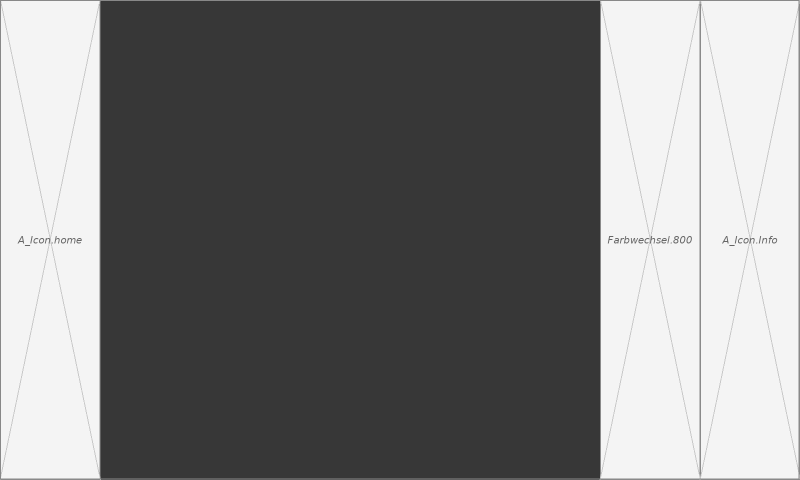
VISUALIZATION Sollwertmenu  // 800x480
    Frame (0,0 800x430)
        shows GWP_Library.Sollwertmenu()
    Frame (0,55 800x121)
        shows GWP_Library.Kachel_Solwertmenu_WG()
        OnMouseClick: change screen: Sollwertmenu_Waermegewinnung
    Frame (0,180 800x121)
        shows GWP_Library.Kachel_Solwertmenu_WP()
        OnMouseClick: change screen: Sollwertmenu_Waermepumpe
    Frame (0,305 800x121)
        shows GWP_Library.Kachel_Solwertmenu_WS()
        OnMouseClick: change screen: Sollwertmenu_Waermesenke
    Frame (0,0 800x480)
        shows Fusszeile_50()
END_VISUALIZATION

// ---- VISUs/Sollwertmenu/Sollwertmenu_Zirk_PU.TcVIS
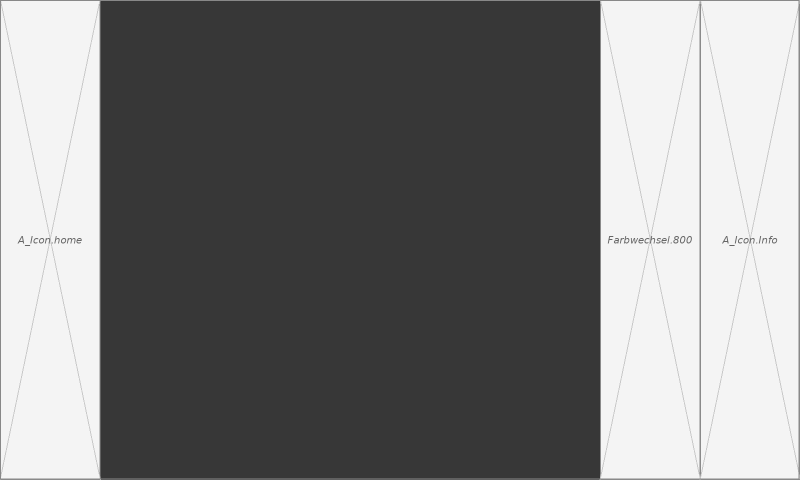
VISUALIZATION Sollwertmenu_Zirk_PU  // 800x480
    Frame (0,0 800x430)
        shows GWP_Library.Sollwertmenu_Zirk_PU()
    Frame (0,55 398x122)
        shows GWP_Library.Kachel_Zirk_PU()
        OnMouseClick: change screen: Zirkulationspumpe_Sollwerte
    Frame (402,55 398x122)
        shows GWP_Library.Kachel_Zirk_PU_Wochenuhr()
        OnMouseClick: change screen: Zirkulationspumpe_CLK_W7_Siebentageprogramm
    Frame (0,0 800x480)
        shows Fusszeile_50()
END_VISUALIZATION

// ---- VISUs/Sollwertmenu/Sollwertmenu_Waermegewinnung.TcVIS
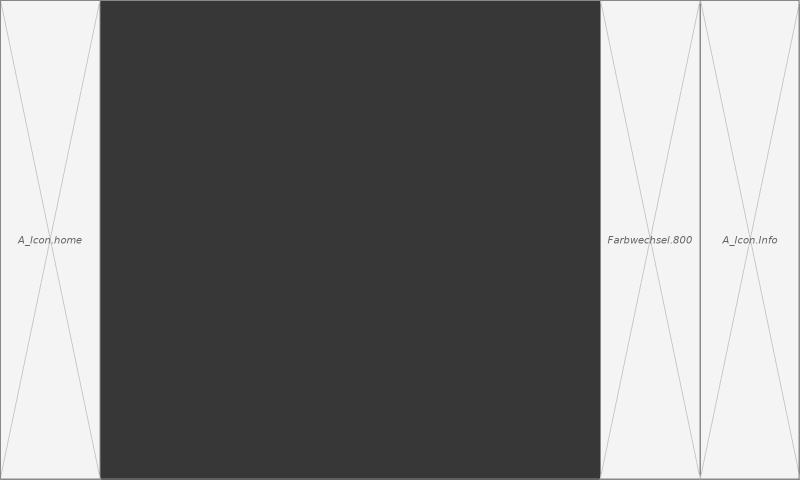
VISUALIZATION Sollwertmenu_Waermegewinnung  // 800x480
    Frame (0,0 800x430)
        shows GWP_Library.Sollwertmenu_Waermegewinnung(FB_KWP_SP_AC_NC := Main.KWP_SP_AC_NC_0, FB_Kreis_3KO := Main.Kreis_3KO_0)
    Frame (0,55 398x121)
        shows GWP_Library.Kachel_PU_VD()
        OnMouseClick: change screen: VD_PU_Sollwerte
    Frame (402,55 398x121)
        shows GWP_Library.Kachel_PU_GW()
        OnMouseClick: change screen: VD_GW_Sollwerte
    Frame (0,304 398x121)
        shows GWP_Library.Kachel_Kaltwasser(FB_Kreis_3KO := Main.Kreis_3KO_0)
        OnMouseClick: change screen: Sollwertmenu_KWP
    Frame (402,179 398x121)
        shows GWP_Library.Kachel_KD_Sollwerte_zuruecksetzen()
        OnMouseClick: change screen: VD_Sollwerte_zuruecksetzen
    Frame (0,179 398x121)
        shows GWP_Library.Kachel_VD_VTL()
        OnMouseClick: change screen: VD_VTL_Sollwerte
    Frame (0,0 800x480)
        shows Fusszeile_50()
END_VISUALIZATION

// ---- VISUs/Sollwertmenu/Sollwertmenu_Waermepumpe.TcVIS
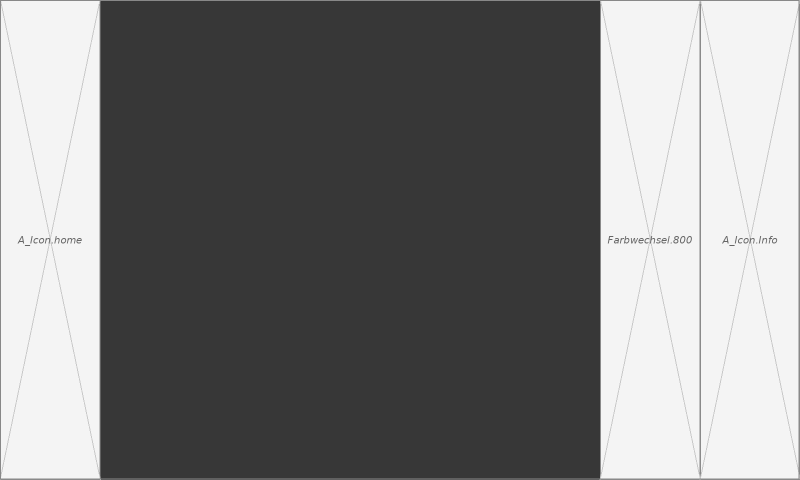
VISUALIZATION Sollwertmenu_Waermepumpe  // 800x480
    Frame (0,0 800x430)
        shows GWP_Library.Sollwertmenu_Waermepumpe()
    Frame (402,55 398x121)
        shows GWP_Library.Kachel_EEV()
        OnMouseClick: change screen: EEv
    Frame (0,179 398x121)
        shows GWP_Library.Kachel_Einsatzgrenzen()
        OnMouseClick: change screen: EG_Innen
    Frame (0,55 398x121)
        shows GWP_Library.Kachel_Allgemein_WP()
        OnMouseClick: change screen: Kreis_3KO_SollwerteAllg
    Frame (0,0 800x480)
        shows Fusszeile_50()
END_VISUALIZATION

// ---- VISUs/Sollwertmenu/Sollwertmenu_KWP.TcVIS
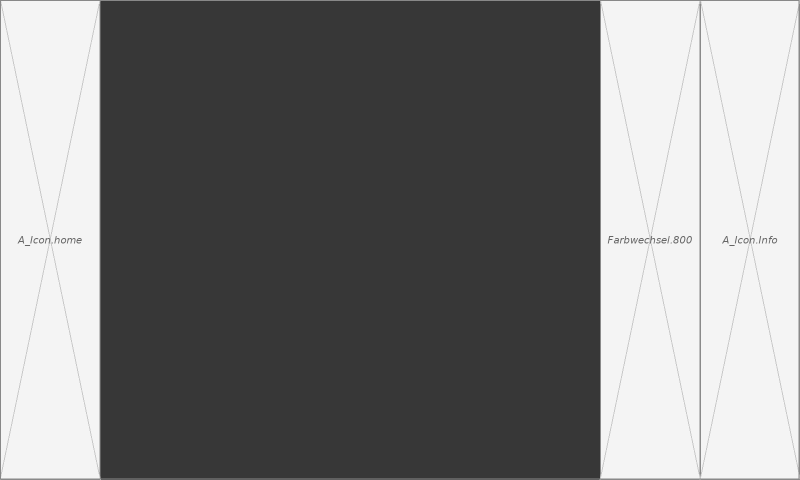
VISUALIZATION Sollwertmenu_KWP  // 800x480
    Frame (0,0 800x430)
        shows GWP_Library.Sollwertmenu_KWP()
    Frame (0,55 398x122)
        shows GWP_Library.Kachel_KWP_Sollwerte(FB_Kreis_3KO := Main.Kreis_3KO_0)
        OnMouseClick: change screen: KWP_SP_AC_NC_Sollwerte
    Frame (402,55 398x122)
        shows GWP_Library.Kachel_KWP_Pumpe()
        OnMouseClick: change screen: KWP_SP_AC_NC_PU_Sollwerte
    Frame (0,179 398x122)
        shows GWP_Library.Kachel_KWP_Tagesuhr_Kuehlkurve()
        OnMouseClick: change screen: KWP_SP_AC_NC_CLK_D
    Frame (402,179 398x121)
        shows GWP_Library.Kachel_KWP_Kuehlkurve()
        OnMouseClick: change screen: KWP_SP_AC_NC_GR_4_ohne_RE
    Frame (0,0 800x480)
        shows Fusszeile_50()
END_VISUALIZATION

// ---- VISUs/Sollwertmenu/Sollwertmenu_Waermesenke.TcVIS
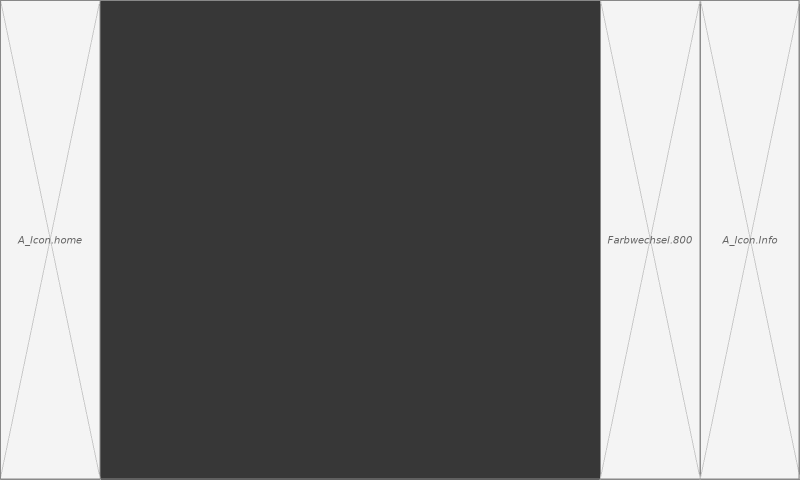
VISUALIZATION Sollwertmenu_Waermesenke  // 800x480
    Frame (0,0 800x430)
        shows GWP_Library.Sollwertmenu_Waermesenke()
    Frame (0,55 398x121)
        shows GWP_Library.Kachel_Hochhaltung()
        OnMouseClick: change screen: Sollwertmenu_KD
    Frame (402,55 398x121)
        shows GWP_Library.Kachel_HWP()
        OnMouseClick: change screen: Sollwertmenu_HWP
    Frame (0,179 398x121)
        shows GWP_Library.Kachel_TWW()
        OnMouseClick: change screen: Sollwertmenu_TWW
    Frame (402,179 398x121)
        shows GWP_Library.Kachel_Zusatzheitzung()
        OnMouseClick: change screen: Zusatzheizung_Sollwerte
    Frame (0,303 398x121)
        shows GWP_Library.Kachel_Zirk_Pumpe()
        OnMouseClick: change screen: Sollwertmenu_Zirk_PU
    Frame (0,55 398x121)
        shows GWP_Library.Kachel_Hochhaltung()
        OnMouseClick: change screen: Sollwertmenu_KD
    Frame (402,55 398x121)
        shows GWP_Library.Kachel_HWP()
        OnMouseClick: change screen: Sollwertmenu_HWP
    Frame (0,179 398x121)
        shows GWP_Library.Kachel_TWW()
        OnMouseClick: change screen: Sollwertmenu_TWW
    Frame (402,179 398x121)
        shows GWP_Library.Kachel_Zirk_PU()
        OnMouseClick: change screen: Sollwertmenu_Zirk_PU
    Frame (0,303 398x121)
        shows GWP_Library.Kachel_Zusatzheitzung()
        OnMouseClick: change screen: Zusatzheizung_Sollwerte
    Frame (0,0 800x480)
        shows Fusszeile_50()
END_VISUALIZATION

// ---- VISUs/Sollwertmenu/Sollwertmenu_KD.TcVIS
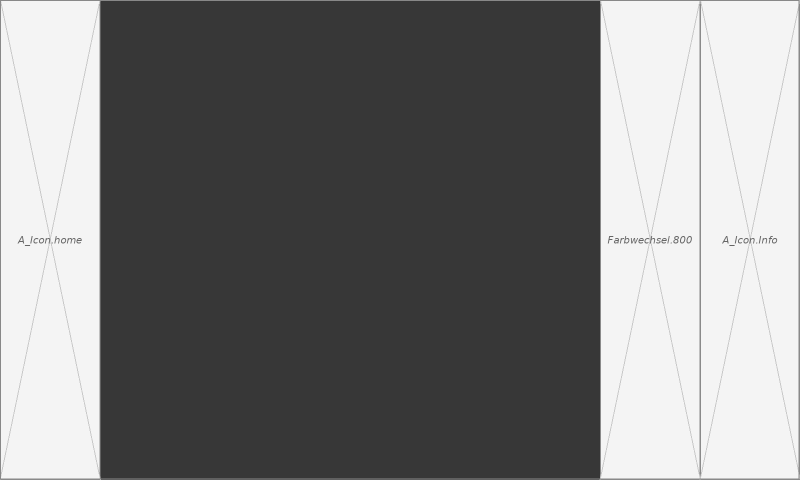
VISUALIZATION Sollwertmenu_KD  // 800x480
    Frame (0,0 800x430)
        shows GWP_Library.Sollwertmenu_KD()
    Frame (0,55 398x121)
        shows GWP_Library.Kachel_KD_Pumpe()
        OnMouseClick: change screen: KD_PU_Sollwerte
    Frame (402,55 398x121)
        shows GWP_Library.Kachel_KD_Ventil()
        OnMouseClick: change screen: KD_VTL_Sollwerte
    Frame (0,179 398x121)
        shows GWP_Library.Kachel_KD_Sollwerte_zuruecksetzen()
        OnMouseClick: change screen: KD_Sollwerte_zuruecksetzen
    Frame (0,0 800x480)
        shows Fusszeile_50()
END_VISUALIZATION

// ---- VISUs/Sollwertmenu/Sollwertmenu_HWP.TcVIS
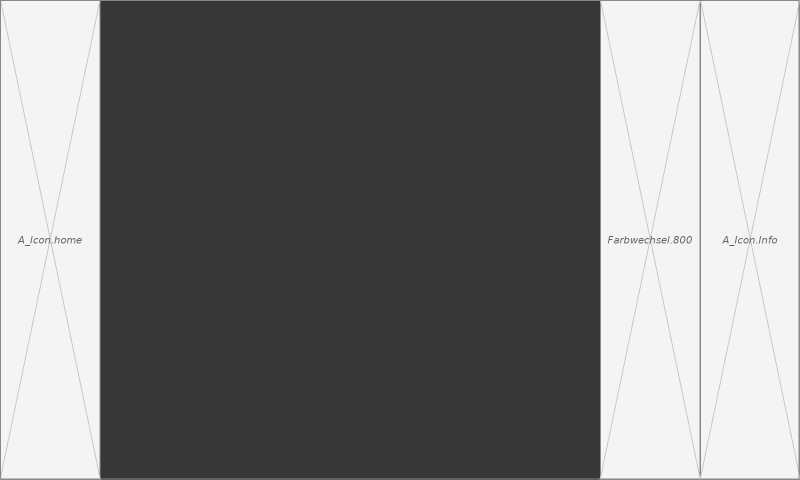
VISUALIZATION Sollwertmenu_HWP  // 800x480
    Frame (0,0 800x430)
        shows GWP_Library.Sollwertmenu_HWP()
    Frame (0,55 398x121)
        shows GWP_Library.Kachel_HWP_Sollwerte(FB_Kreis_3KO := Main.Kreis_3KO_0)
        OnMouseClick: change screen: HWP_SP_Sollwerte
    Frame (402,55 398x121)
        shows GWP_Library.Kachel_HWP_Tagesuhr_Heizkurve()
        OnMouseClick: change screen: HWP_SP_CLK_D
    Frame (0,179 398x121)
        shows GWP_Library.Kachel_HWP_Heizkurve()
        OnMouseClick: change screen: HWP_SP_GR_4_ohne_RE
    Frame (0,0 800x480)
        shows Fusszeile_50()
END_VISUALIZATION

// ---- VISUs/Sollwertmenu/Sollwertmenu_TWW.TcVIS
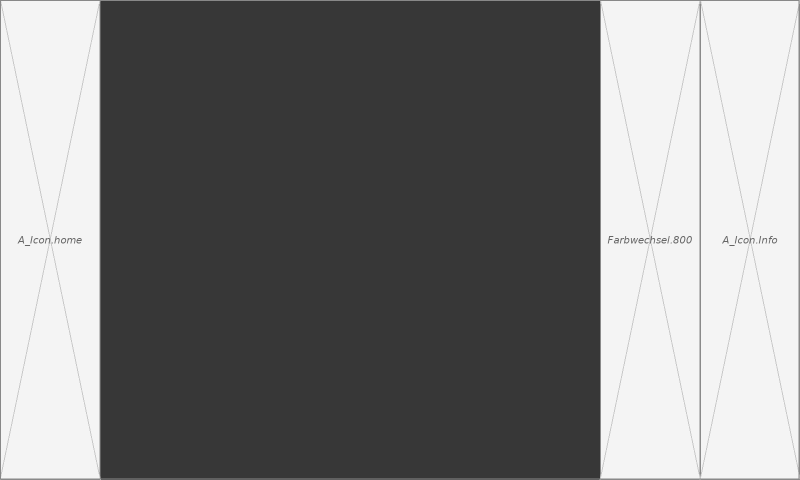
VISUALIZATION Sollwertmenu_TWW  // 800x480
    Frame (0,0 800x430)
        shows GWP_Library.Sollwertmenu_TWW()
    Frame (0,55 398x121)
        shows GWP_Library.Kachel_TWW_SP_Sollwerte()
        OnMouseClick: change screen: TWW_SP_Sollwerte
    Frame (402,55 398x121)
        shows GWP_Library.Kachel_TWW_SP_Pumpe()
        OnMouseClick: change screen: TWW_SP_PU_Sollwerte
    Frame (0,179 398x121)
        shows GWP_Library.Kachel_TWW_SP_Zwangsladung_1()
        OnMouseClick: change screen: TWW_SP_CLK_I_Zwangsladung_1
    Frame (402,179 398x121)
        shows GWP_Library.Kachel_TWW_SP_Zwangsladung_2()
        OnMouseClick: change screen: TWW_SP_CLK_I_Zwangsladung_2
    Frame (0,0 800x480)
        shows Fusszeile_50()
END_VISUALIZATION

// ---- VISUs/Test_Login.TcVIS
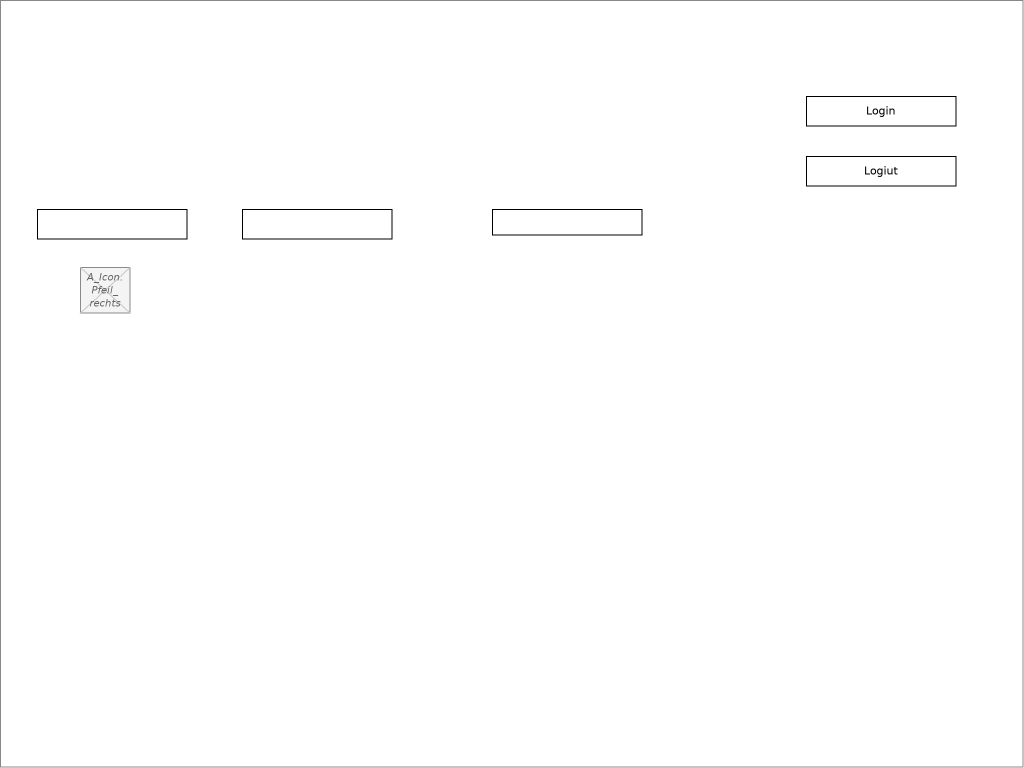
VISUALIZATION Test_Login  // 1024x768
VAR_IN_OUT
	FB_AI_8:AI_8;
END_VAR
    Rectangle (37,209 150x30)
        OnMouseClick: change screen: Home
    Rectangle (242,209 150x30)
        OnMouseClick: change screen: Home
    Rectangle (492,209 150x26)
    Rectangle (806,96 150x30), "Login"
        OnMouseClick: VisuUserMgmt Type=Login
    Rectangle (806,156 150x30), "Logiut"
        OnMouseClick: VisuUserMgmt Type=Logout
    Image (80,267 50x46), image: A_Icon.Pfeil_rechts
        OnMouseClick: execute { Visu.i_Frame_VD_Index:=4; }
END_VISUALIZATION

// ---- VISUs/Testkachel.TcVIS
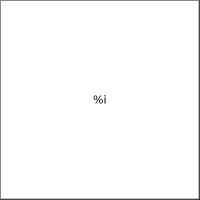
VISUALIZATION Testkachel  // 200x200
VAR_IN_OUT
	FB_DI_16:DI_16;
END_VAR
var_input
	s_Titel:STRING;
END_VAR
    Rectangle (0,0 200x200), "%i", text variable: s_Titel
END_VISUALIZATION
